FUNCTION alg_a_Dresetled : BOOL
VAR_INPUT
	state: STATE;
END_VAR

alg_a_Dresetled := alg_M_example_controller_a_Dresetled(state);

END_FUNCTION

(* stored: Version 1.1.0.1, ProductVersion 3.1.4022.18
   POU alg_a_Dresetled: Id {a6fa8f4b-597a-4b34-adc4-f882e49969c7}, SpecialFunc None *)
